FUNCTION_BLOCK Bx1CoverFailsafe (* BX1 cover output SAFE-START gate. On INIT/cold/warm start it forces CoverPNP_Hr to HOME (ToWork=0, ToHome=1) and CoverPNP_Vr/Gripper de-energised, and HOLDS that until the Hr at-home sensor is TRUE AND the actuator is no longer commanding Work, then passes the live cover coils through. Guarantees cover_hr can never auto-energise Work on deploy/login/restart (whenever the logic runs) and actively drives it home if left at Work. NOTE: runtime gate only - does NOT act on EAE Clean/STOP/fault (logic stops, output word frozen). Homing while stopped needs the TM3BC coupler ToHome fallback (word 16#0002), a coupler-side setting outside the Mapper. *)
  (* Standard: 61499-2 *)
  (* Version 0.1, 6/30/2026, easensoy, WMG, BX1 CoverPNP_Hr swivel-collision safe-start *)
  PACKAGE Main;
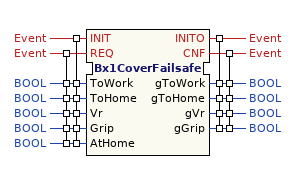
  EVENT_INPUT
    INIT WITH ToWork, ToHome, Vr, Grip, AtHome; (* Arm safe-start: force the covers to the safe home pattern *)
    REQ WITH ToWork, ToHome, Vr, Grip, AtHome; (* Recompute the gated output bits for this scan *)
  END_EVENT
  EVENT_OUTPUT
    INITO WITH gToWork, gToHome, gVr, gGrip; (* Safe-start armed *)
    CNF WITH gToWork, gToHome, gVr, gGrip; (* Gated output bits ready *)
  END_EVENT
  VAR_INPUT
    ToWork : BOOL; (* Live CoverPNP_Hr advance coil (OutputToWork) *)
    ToHome : BOOL; (* Live CoverPNP_Hr retract coil (OutputToHome) *)
    Vr : BOOL; (* Live CoverPNP_Vr work coil *)
    Grip : BOOL; (* Live CoverPnp_Gripper work coil *)
    AtHome : BOOL; (* CoverPNP_Hr at-home sensor (input word bit0) *)
  END_VAR
  VAR_OUTPUT
    gToWork : BOOL; (* Gated Hr advance bit (forced FALSE while safe-start is armed) *)
    gToHome : BOOL; (* Gated Hr retract bit (forced TRUE while safe-start is armed = drive home) *)
    gVr : BOOL; (* Gated Vr bit (forced FALSE while armed) *)
    gGrip : BOOL; (* Gated gripper bit (forced FALSE while armed) *)
  END_VAR
  VAR
    safe : BOOL; (* TRUE = safe-start armed (force CoverPNP_Hr home) *)
  END_VAR
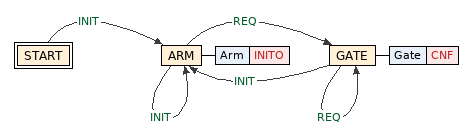
  EC_STATES
    START; (* Initial State *)
    ARM : Arm -> INITO; (* Arm safe-start (force home) *)
    GATE : Gate -> CNF; (* Gate each scan until home reached *)
  END_STATES
  EC_TRANSITIONS
    START TO ARM := INIT;
    ARM TO ARM := INIT;
    ARM TO GATE := REQ;
    GATE TO ARM := INIT;
    GATE TO GATE := REQ;
  END_TRANSITIONS
  ALGORITHM Arm IN ST: (* Arm safe-start: force CoverPNP_Hr to HOME, all other cover coils OFF *)
safe := TRUE;
gToWork := FALSE;
gToHome := TRUE;
gVr := FALSE;
gGrip := FALSE;
  END_ALGORITHM
  ALGORITHM Gate IN ST: (* Hold the safe home command until Hr at-home AND the actuator is no longer commanding Work (else the latched ToWork coil would drive the cover straight back to Work on release), then pass the live cover coils through *)
IF AtHome AND NOT ToWork THEN
	safe := FALSE;
END_IF;
IF safe THEN
	gToWork := FALSE;
	gToHome := TRUE;
	gVr := FALSE;
	gGrip := FALSE;
ELSE
	gToWork := ToWork;
	gToHome := ToHome;
	gVr := Vr;
	gGrip := Grip;
END_IF;
  END_ALGORITHM
END_FUNCTION_BLOCK
